// TIA Portal V19 export
VAR_GLOBAL   // PLC tag table "S71200IDevice"
   "Out to 1200" AT %QW100 : Int;
   PB_Green_from_1200 AT %I100.0 : Bool;
   PB_Blue_from_1200 AT %I100.1 : Bool;
   POT_from_1200 AT %IW102 : Word;
END_VAR
